// TIA Portal V20 export
TYPE "typeSequenceControlNodeHomeCheck_transferPnPRight"
// stored: Namespace Unit1.Em5
   STRUCT
      waitPosPartNoDetect { ExternalWritable := 'False'} : Bool;
      waitPosPartDetect { ExternalWritable := 'False'} : Bool;
      hipotThicknessPosPartNoDetect { ExternalWritable := 'False'} : Bool;
      hipotThicknessPosPartDetect { ExternalWritable := 'False'} : Bool;
      visionPosPartNoDetect { ExternalWritable := 'False'} : Bool;
      visionPosPartDetect { ExternalWritable := 'False'} : Bool;
      laserMarkPosPartNoDetect { ExternalWritable := 'False'} : Bool;
      laserMarkPosPartDetect { ExternalWritable := 'False'} : Bool;
      weightCheckPosPartNoDetect { ExternalWritable := 'False'} : Bool;
      weightCheckPosPartDetect { ExternalWritable := 'False'} : Bool;
      defaultPosPartDetect : Bool;
      defaultPosPartNoDetect : Bool;
   END_STRUCT;
END_TYPE
